{attribute 'qualified_only'}
{attribute 'strict'}
TYPE
    eInspectionGroupTests :
    (
        Inspect         := 10,
        GetResult       := 20,
        OnFailCarryOn   := 40,
        OnFailRetry     := 50,
        OnFailTerminate := 60,
		OnFailDiaglog   := 70
    );
END_TYPE

(* stored: Version 1.1.0.1, ProductVersion 3.1.4024.9
   DUT eInspectionGroupTests: Id {cab3fe3a-81a0-04f9-0588-68a8f9a8d44a} *)
